SUBAPPLICATION AR_Timeout_Zero (* Fendt-Schaltung (4diac_training1 Uebung_074_AUI.SUB): liefert IN0 unveraendert, ausser G (i.d.R. IA_*.TIMEOUT - echter Kommunikationsausfall) ist TRUE, dann 0.0 statt des sonst einfach eingefrorenen letzten Werts. *)
  (* Standard: 61499-2; Description: Copyright (c) 2026 Meisterschulen am Ostbahnhof This program and the accompanying materials are made available under the terms of the Eclipse Public License 2.0 which is available at https://www.eclipse.org/legal/epl-2.0/ SPDX-License-Identifier: EPL-2.0 *)
  (* Version 1.1, 2026-09-16, Franz Höpfinger, Meisterschulen am Ostbahnhof, Nach MyLib_AX-1.0.0::sys verschoben (Franz) - generischer Baustein, gehoert nicht in den TECU-spezifischen Ordner. *)
  (* Version 1.0, 2026-09-16, Franz Höpfinger, Meisterschulen am Ostbahnhof, Herausgeloest (Franz: 'AR_AX_SEL_AR initval_AR=0 kann eine SUB sein, das haben wir ja OFT') - AR_AX_SEL_AR + initval_AR(0.0) wurde in TECU_RPTO/TECU_FPTO/TECU_COGSOG/TECU_GBSD/TECU_WBSD/TECU_VDS/TECU_FHS/TECU_RHS/TECU_MSS jeweils einzeln verdrahtet, jetzt ein wiederverwendbarer Baustein. *)
  PACKAGE MyLib::sys;
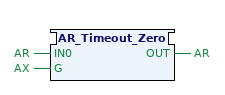
  SOCKETS
    IN0 : adapter::types::unidirectional::AR; (* Live-Wert, z.B. FIELDBUS_*_SCALED.OUT *)
    G : adapter::types::unidirectional::AX; (* TRUE = Timeout, liefert 0.0 statt IN0 *)
  END_SOCKETS
  PLUGS
    OUT : adapter::types::unidirectional::AR; (* IN0, oder 0.0 bei G=TRUE *)
  END_PLUGS
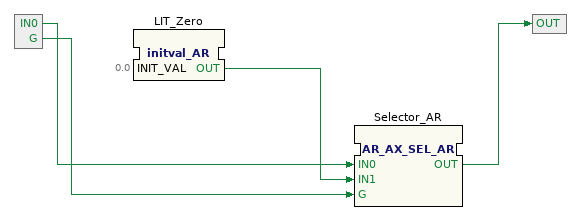
  FBS
    LIT_Zero : adapter::types::unidirectional::AR::initval::initval_AR(INIT_VAL := 0.0);
    Selector_AR : adapter::iec61131::selection::AR_AX_SEL_AR;
  END_FBS
  ADAPTER_CONNECTIONS
    IN0 TO Selector_AR.IN0;
    LIT_Zero.OUT TO Selector_AR.IN1;
    G TO Selector_AR.G;
    Selector_AR.OUT TO OUT;
  END_CONNECTIONS
END_SUBAPPLICATION
